INTERFACE I_DriveReverse EXTENDS I_Drive

METHOD SwitchReverseOff : BOOL
VAR_INPUT
END_VAR
END_METHOD

METHOD SwitchReverseON : BOOL
VAR_INPUT
END_VAR
END_METHOD

END_INTERFACE

(* stored: Version 1.1.0.1, ProductVersion 3.1.4024.12
   Itf I_DriveReverse: Id {7e6fb88b-ab30-49e9-aab8-c2339bf84641}
   Method SwitchReverseOff: Id {de8545cc-c9b7-4f9d-bf20-d93d9b164788}
   Method SwitchReverseON: Id {f9735176-34e5-45e5-8a15-bb554486a2c6} *)
